// Mitsubishi GX Works2 project: 240402_인칭회로   PLC: Q03UDV

PROGRAM MAIN
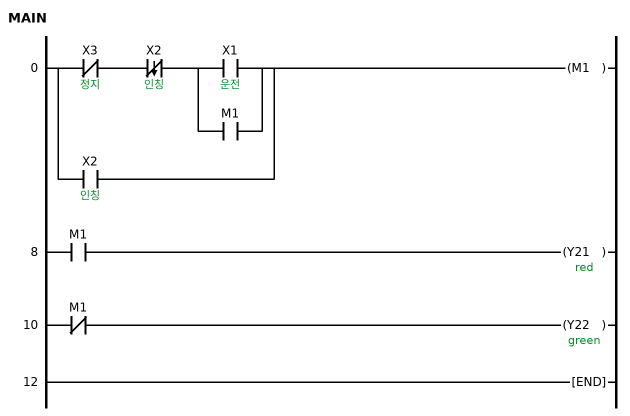
0     LDI     X3  ; 정지
      ANDFI   X2  ; 인칭
      LD      X1  ; 운전
      OR      M1
      ANB
      OR      X2  ; 인칭
      OUT     M1
8     LD      M1
      OUT     Y21  ; red
10    LDI     M1
      OUT     Y22  ; green
12    END
END_PROGRAM
